FUNCTION_BLOCK TransportActuatorGripper EXTENDS ZEquipment.ActuatorDigitalBiLsPlusMinus

METHOD PUBLIC CloseAsync
VAR_INPUT
  startToken : ZCore.IStartToken;
END_VAR
MoveMinusAsync(startToken:=startToken);
END_METHOD

METHOD PUBLIC IsClosed : BOOL
VAR_INPUT
END_VAR
IsClosed := IsAtMinus();
END_METHOD

METHOD PUBLIC IsOpen : BOOL
VAR_INPUT
END_VAR
IsOpen := IsAtPlus();
END_METHOD

METHOD PUBLIC OpenAsync
VAR_INPUT
  startToken : ZCore.IStartToken;
END_VAR
MovePlusAsync(startToken:=startToken);
END_METHOD

END_FUNCTION_BLOCK

(* stored: Version 1.1.0.1
   POU TransportActuatorGripper: Id {d0b6f853-c65d-477e-8967-40d5ae4bc598}, SpecialFunc None
   Method CloseAsync: Id {e9d276c1-1f6d-43ac-90c6-7d03811f9914}
   Method IsClosed: Id {b47c364c-42d5-49c7-ad2d-d40e4562feca}
   Method IsOpen: Id {2150f9f5-3664-463d-897f-f6c2015e9768}
   Method OpenAsync: Id {a0bee3d9-076e-4b9b-9b2b-8e83df724b0e} *)
